# EPICS substitutions: epics-driver/picoApp/Db/pico8_chan_alias.substitutions
#dbLoadRecords("../../db/pico8_chan_alias.db", "P=DIAG_MTCA01:PICO3_CH0:,A=FE_SCS2:EMS_D0718Y:")

file "pico8_chan_alias.template"
{
{P="\$(P)", A="\$(A)"}
}

file "pico8_cap_float_alias.template"
{
{P="\$(P)AVG", A="\$(A)AVG"}
{P="\$(P)ASTD",A="\$(A)ASTD"}
{P="\$(P)MIN", A="\$(A)MIN"}
{P="\$(P)MAX", A="\$(A)MAX"}
{P="\$(P)STD", A="\$(A)STD"}
}
